FUNCTION_BLOCK FB_EnduranceInfraredPyrometer
VAR_INPUT
END_VAR
VAR_OUTPUT
END_VAR
VAR
	_tcpIp	: ZigaLibs_TcpIp.FB_TcpIpCommControl;
END_VAR

END_FUNCTION_BLOCK

(* stored: Version 1.1.0.1, ProductVersion 3.1.4024.15
   POU FB_EnduranceInfraredPyrometer: Id {6a4433dd-bb61-0fcc-078b-e154b0f6633d}, SpecialFunc None *)
